FUNCTION_BLOCK FB_EventsManager
VAR_INPUT
    // Presentation-only warning classification; does not request Fault/Stop.
    aWarningEvents : ARRAY[0..4, 0..100] OF BOOL;
	bPulse					: BOOL;
	bDataWritedInCSV		: BOOL;
	nArraySize				: DINT;
	bMachineMessage			: STRING;
	eMachineState 			: E_MachineState;
END_VAR
VAR_OUTPUT
    bMachineFault            : BOOL;
    bCycleStopRequest        : BOOL;
    sSystemDate              : STRING(10);
    sSystemTime              : STRING(8);
	astActiveEvents			: ARRAY [0..50] OF ST_ActiveEvents;
	astEventsHistory		: ARRAY[0..200] OF ST_EventsHistory;
END_VAR
VAR
    aWarningConditionSeen : ARRAY[0..4, 0..100] OF BOOL;
	i								: ARRAY [0..1] OF DINT;
	j								: ARRAY [0..1] OF DINT;
	m								: ARRAY [0..3] OF DINT;
	k								: ARRAY [0..1] OF DINT;
	l								: DINT;
	n								: DINT;
	
	bEventsAssigmentSignal			: BOOL		:= TRUE;
    bStationFaultCondition   : BOOL;
    bStationStopCondition    : BOOL;

    // Local IPC clock used internally for event-history timestamps.
    fbLocalSystemTime        : FB_LocalSystemTime;
END_VAR

VAR_IN_OUT
	
	stStationEvents			: ARRAY[0..4] OF ST_StationEvents;
	stEventsAssigment		: ST_EventsAssigmentGeneral;
	bResetFaults			: BOOL;
	
END_VAR

UpdateSystemDateTime();

ACT_FaultTrig();

ACT_EventTextAssigment();

ACT_ActiveEvents_DataHistory();

// Row zero is permanently reserved for the operational instruction.
astActiveEvents[0].sEventTex := bMachineMessage;
astActiveEvents[0].sType := 'Message';
astActiveEvents[0].abType := 3;
astActiveEvents[0].sSolution := '';

ACTION ACT_ActiveEvents_DataHistory:
// ============================================================================
// ACTIVE EVENTS AND EVENT HISTORY
// ============================================================================
//
// astActiveEvents[0]:
//     Reserved exclusively for the current machine message.
//
// astActiveEvents[1..50]:
//     Active Faults and Cycle Stop Requests.
//
// astEventsHistory:
//     Complete event history.
//
// EVENT BEHAVIOUR:
//
// MESSAGE:
//     - Operator instruction.
//     - Displayed only through astActiveEvents[0].
//     - Never added to rows 1..50.
//
// FAULT:
//     - Latched individually through bActive.
//     - Displayed only while the machine is in Fault.
//     - Remains latched after the live condition disappears.
//     - Cleared by Reset only after bEventFlag is FALSE.
//
// CYCLE STOP REQUEST:
//     - Latched individually through bActive.
//     - Displayed in any machine state.
//     - Remains visible after the live condition disappears.
//     - Cleared by Reset only after bEventFlag is FALSE.
//
// bEventFlag:
//     Live condition.
//
// bActive:
//     Individual event presentation latch.
//
// ============================================================================


IF bPulse THEN

    // ------------------------------------------------------------------------
    // REBUILD ACTIVE EVENT GRID
    // ------------------------------------------------------------------------
    // Row 0 is intentionally preserved because it contains the current
    // machine instruction/message.
    // ------------------------------------------------------------------------

    FOR l := 1 TO 50 DO

        astActiveEvents[l].sEventTex := '';
        astActiveEvents[l].sType := '';
        astActiveEvents[l].abType := 0;
        astActiveEvents[l].sSolution := '';

    END_FOR


    // Rows 1..50 are used for Faults and Alerts.
    l := 0;


    // ------------------------------------------------------------------------
    // SCAN ALL STATION EVENTS
    // ------------------------------------------------------------------------

    FOR k[0] := 0 TO nArraySize DO

        FOR k[1] := 0 TO 100 DO


            // =================================================================
            // FAULT
            // =================================================================

            IF stStationEvents[k[0]].aEvents[k[1]].bFault THEN


                // -------------------------------------------------------------
                // NEW FAULT DETECTED
                // -------------------------------------------------------------
                // Register in history only once, when the live condition
                // activates an event that was not already latched.
                // -------------------------------------------------------------

                IF stStationEvents[k[0]].aEvents[k[1]].bEventFlag
                    AND NOT stStationEvents[k[0]].aEvents[k[1]].bActive
                THEN

                    // Shift history.
                    FOR n := 200 TO 1 BY -1 DO

                        astEventsHistory[n] :=
                            astEventsHistory[n - 1];

                    END_FOR


                    // Insert newest event.
                    astEventsHistory[0].sEventTex :=
                        stStationEvents[k[0]].aEvents[k[1]].bEventTextHMI;

                    astEventsHistory[0].sType :=
                        'Fault';

                    astEventsHistory[0].abType :=
                        1;

                    astEventsHistory[0].sDate :=
                        sSystemDate;

                    astEventsHistory[0].sTime :=
                        sSystemTime;


                    // Latch the individual event.
                    stStationEvents[k[0]].aEvents[k[1]].bActive :=
                        TRUE;

                END_IF


                // -------------------------------------------------------------
                // RESET FAULT LATCH
                // -------------------------------------------------------------
                // Reset is allowed to clear the individual event only after
                // the originating fault condition has disappeared.
                // -------------------------------------------------------------

                IF bResetFaults
                    AND NOT stStationEvents[k[0]].aEvents[k[1]].bEventFlag
                THEN

                    stStationEvents[k[0]].aEvents[k[1]].bActive :=
                        FALSE;

                END_IF


                // -------------------------------------------------------------
                // ACTIVE GRID
                // -------------------------------------------------------------
                // Faults are shown only while the machine itself is in Fault.
                //
                // bActive allows the original cause to remain displayed after
                // bEventFlag has returned FALSE, until the operator resets.
                // -------------------------------------------------------------

                IF stStationEvents[k[0]].aEvents[k[1]].bActive
                    AND eMachineState = E_MachineState.Fault
                THEN

                    IF l < 50 THEN

                        l := l + 1;

                        astActiveEvents[l].sEventTex :=
                            stStationEvents[k[0]].aEvents[k[1]].bEventTextHMI;

                        astActiveEvents[l].sType :=
                            'Fault';

                        astActiveEvents[l].abType :=
                            1;

                        astActiveEvents[l].sSolution :=
                            stStationEvents[k[0]].aEvents[k[1]].sSolution;

                    END_IF

                END_IF



            // =================================================================
            // CYCLE STOP REQUEST / ALERT
            // =================================================================

            ELSIF stStationEvents[k[0]].aEvents[k[1]].bCycleStopRequest THEN


                // -------------------------------------------------------------
                // NEW ALERT DETECTED
                // -------------------------------------------------------------

                IF stStationEvents[k[0]].aEvents[k[1]].bEventFlag
                    AND NOT stStationEvents[k[0]].aEvents[k[1]].bActive
                THEN

                    // Shift history.
                    FOR n := 200 TO 1 BY -1 DO

                        astEventsHistory[n] :=
                            astEventsHistory[n - 1];

                    END_FOR


                    // Insert newest event.
                    astEventsHistory[0].sEventTex :=
                        stStationEvents[k[0]].aEvents[k[1]].bEventTextHMI;

                    astEventsHistory[0].sType :=
                        'Cycle Stop Request';

                    astEventsHistory[0].abType :=
                        2;

                    astEventsHistory[0].sDate :=
                        sSystemDate;

                    astEventsHistory[0].sTime :=
                        sSystemTime;


                    // Latch the individual Alert.
                    stStationEvents[k[0]].aEvents[k[1]].bActive :=
                        TRUE;

                END_IF


                // -------------------------------------------------------------
                // RESET ALERT LATCH
                // -------------------------------------------------------------
                // The Alert remains displayed after the live condition has
                // disappeared and is acknowledged by Reset.
                // -------------------------------------------------------------

                IF bResetFaults
                    AND NOT stStationEvents[k[0]].aEvents[k[1]].bEventFlag
                THEN

                    stStationEvents[k[0]].aEvents[k[1]].bActive :=
                        FALSE;

                END_IF


                // -------------------------------------------------------------
                // ACTIVE GRID
                // -------------------------------------------------------------
                // Alerts may be shown in any machine state.
                // -------------------------------------------------------------

                IF stStationEvents[k[0]].aEvents[k[1]].bActive THEN

                    IF l < 50 THEN

                        l := l + 1;

                        astActiveEvents[l].sEventTex :=
                            stStationEvents[k[0]].aEvents[k[1]].bEventTextHMI;

                        astActiveEvents[l].sType :=
                            'Cycle Stop Request';

                        astActiveEvents[l].abType :=
                            2;

                        astActiveEvents[l].sSolution :=
                            stStationEvents[k[0]].aEvents[k[1]].sSolution;

                    END_IF

                END_IF



            // =================================================================
            // MESSAGE
            // =================================================================
            //
            // Messages are instructions for the operator.
            //
            // They are NOT inserted into astActiveEvents[1..50].
            // Row 0 remains exclusively responsible for the current machine
            // instruction through sMachineMessage.
            //
            // bActive is not used as an operator-reset latch for Messages.
            // =================================================================

            // Resettable warnings use the existing Alert icon (abType=2).
            // The raw condition rearms history; bActive retains display until Reset.
            // Acknowledging a held condition must not re-create the warning.
            ELSIF aWarningEvents[k[0], k[1]] THEN

                IF stStationEvents[k[0]].aEvents[k[1]].bEventFlag
                    AND NOT aWarningConditionSeen[k[0], k[1]]
                THEN
                    FOR n := 200 TO 1 BY -1 DO
                        astEventsHistory[n] := astEventsHistory[n - 1];
                    END_FOR
                    astEventsHistory[0].sEventTex :=
                        stStationEvents[k[0]].aEvents[k[1]].bEventTextHMI;
                    astEventsHistory[0].sType := 'Warning';
                    astEventsHistory[0].abType := 2;
                    astEventsHistory[0].sDate := sSystemDate;
                    astEventsHistory[0].sTime := sSystemTime;
                    stStationEvents[k[0]].aEvents[k[1]].bActive := TRUE;
                END_IF

                aWarningConditionSeen[k[0], k[1]] :=
                    stStationEvents[k[0]].aEvents[k[1]].bEventFlag;
                // Live owner-latched warnings cannot be acknowledged by machine Reset.
                IF stStationEvents[k[0]].aEvents[k[1]].bPersistentMessage THEN
                    stStationEvents[k[0]].aEvents[k[1]].bActive :=
                        stStationEvents[k[0]].aEvents[k[1]].bEventFlag;
                ELSIF bResetFaults THEN
                    stStationEvents[k[0]].aEvents[k[1]].bActive := FALSE;
                END_IF

                IF stStationEvents[k[0]].aEvents[k[1]].bActive AND (l < 50) THEN
                    l := l + 1;
                    astActiveEvents[l].sEventTex :=
                        stStationEvents[k[0]].aEvents[k[1]].bEventTextHMI;
                    astActiveEvents[l].sType := 'Warning';
                    astActiveEvents[l].abType := 2;
                    astActiveEvents[l].sSolution :=
                        stStationEvents[k[0]].aEvents[k[1]].sSolution;
                END_IF

            ELSIF stStationEvents[k[0]].aEvents[k[1]].bMessage THEN


                // -------------------------------------------------------------
                // OPTIONAL MESSAGE HISTORY
                // -------------------------------------------------------------
                // Preserve the existing ability to register message events in
                // history, but rearm them automatically when their condition
                // disappears because Messages do not require operator Reset.
                // -------------------------------------------------------------

                IF stStationEvents[k[0]].aEvents[k[1]].bEventFlag
                    AND NOT stStationEvents[k[0]].aEvents[k[1]].bActive
                THEN

                    FOR n := 200 TO 1 BY -1 DO

                        astEventsHistory[n] :=
                            astEventsHistory[n - 1];

                    END_FOR


                    astEventsHistory[0].sEventTex :=
                        stStationEvents[k[0]].aEvents[k[1]].bEventTextHMI;

                    astEventsHistory[0].sType :=
                        'Message';

                    astEventsHistory[0].abType :=
                        3;

                    astEventsHistory[0].sDate :=
                        sSystemDate;

                    astEventsHistory[0].sTime :=
                        sSystemTime;


                    stStationEvents[k[0]].aEvents[k[1]].bActive :=
                        TRUE;

                END_IF


                // Messages automatically rearm when their live condition ends.
                IF NOT stStationEvents[k[0]].aEvents[k[1]].bEventFlag THEN

                    stStationEvents[k[0]].aEvents[k[1]].bActive :=
                        FALSE;

                END_IF

                // Live message: shown in Active Events while the condition is
                // TRUE and cannot be acknowledged/reset by the operator.
                IF stStationEvents[k[0]].aEvents[k[1]].bPersistentMessage
                    AND stStationEvents[k[0]].aEvents[k[1]].bEventFlag
                THEN

                    IF l < 50 THEN
                        l := l + 1;
                        astActiveEvents[l].sEventTex :=
                            stStationEvents[k[0]].aEvents[k[1]].bEventTextHMI;
                        astActiveEvents[l].sType := 'Message';
                        astActiveEvents[l].abType := 3;
                        astActiveEvents[l].sSolution :=
                            stStationEvents[k[0]].aEvents[k[1]].sSolution;
                    END_IF

                END_IF


            END_IF


        END_FOR

    END_FOR


END_IF
END_ACTION

ACTION ACT_EventTextAssigment:

FOR j[0] := 0 TO nArraySize DO
	
	FOR j[1] := 0 TO 100 DO 
		
		IF stStationEvents[j[0]].aEvents[j[1]].bFault THEN
			
			m[0]											:= m[0]+1;
			
			stStationEvents[j[0]].aEvents[j[1]].bEventTextHMI	:= 		CONCAT( STR1 := 'N ', STR2 := 
																CONCAT( STR1 := DINT_TO_STRING(m[0]), str2 := 
																CONCAT( STR1 :='-Station' , STR2 := 
																CONCAT( STR1 := DINT_TO_STRING(j[0]), STR2 := 
																CONCAT( STR1 :=' - ', str2 := stStationEvents[j[0]].aEvents[j[1]].bEventText )))));
			stStationEvents[j[0]].aEvents[j[1]].bAssignedID	:= 	m[0];				
			
			//EVENTS ASSIGMENT
			stEventsAssigment.astFaultEvents[m[0]].sEventText	:= stStationEvents[j[0]].aEvents[j[1]].bEventTextHMI;
			stEventsAssigment.astFaultEvents[m[0]].sSolution	:= stStationEvents[j[0]].aEvents[j[1]].sSolution;
			
		ELSIF stStationEvents[j[0]].aEvents[j[1]].bCycleStopRequest THEN
		
			m[2]											:= m[2]+1;	
			
			stStationEvents[j[0]].aEvents[j[1]].bEventTextHMI	:= 		CONCAT( STR1 := 'N ', STR2 := 
																CONCAT( STR1 := DINT_TO_STRING(m[2]), str2 := 
																CONCAT( STR1 :='-Station' , STR2 := 
																CONCAT( STR1 := DINT_TO_STRING(j[0]), STR2 := 
																CONCAT( STR1 :=' - ', str2 := stStationEvents[j[0]].aEvents[j[1]].bEventText )))));
			stStationEvents[j[0]].aEvents[j[1]].bAssignedID	:= 	m[2];													

			//EVENTS ASSIGMENT
			stEventsAssigment.astCycleStopRequestEvents[m[2]].sEventText	:= stStationEvents[j[0]].aEvents[j[1]].bEventTextHMI;
			stEventsAssigment.astCycleStopRequestEvents[m[2]].sSolution	:= stStationEvents[j[0]].aEvents[j[1]].sSolution;
			
		ELSIF stStationEvents[j[0]].aEvents[j[1]].bMessage THEN
			
			m[3]											:= m[3]+1;
			
			stStationEvents[j[0]].aEvents[j[1]].bEventTextHMI	:= 		CONCAT( STR1 := 'N ', STR2 := 
																CONCAT( STR1 := DINT_TO_STRING(m[3]), str2 := 
																CONCAT( STR1 :='-Station' , STR2 := 
																CONCAT( STR1 := DINT_TO_STRING(j[0]), STR2 := 
																CONCAT( STR1 :=' - ', str2 := stStationEvents[j[0]].aEvents[j[1]].bEventText )))));
			stStationEvents[j[0]].aEvents[j[1]].bAssignedID	:= 	m[3];													
				
			//EVENTS ASSIGMENT
			stEventsAssigment.astMessage[m[3]].sEventText	:= stStationEvents[j[0]].aEvents[j[1]].bEventTextHMI;
			stEventsAssigment.astMessage[m[3]].sSolution	:= stStationEvents[j[0]].aEvents[j[1]].sSolution;	
			
		END_IF
		
	END_FOR
	
	
END_FOR
j[0]														:= 0;
j[1]														:= 0;
m[0]														:= 0;
m[1]														:= 0;
m[2]														:= 0;
m[3]														:= 0;
END_ACTION

ACTION ACT_FaultTrig:
// Deterministic station aggregation. Classification is fixed in each point;
// bEventFlag is the live condition. Station flags are latched until Reset.
bMachineFault := FALSE;
bCycleStopRequest := FALSE;

FOR i[0] := 0 TO nArraySize DO
    bStationFaultCondition := FALSE;
    bStationStopCondition := FALSE;

    FOR i[1] := 0 TO 100 DO
        bStationFaultCondition := bStationFaultCondition
            OR (stStationEvents[i[0]].aEvents[i[1]].bFault
                AND stStationEvents[i[0]].aEvents[i[1]].bEventFlag);

        bStationStopCondition := bStationStopCondition
            OR (stStationEvents[i[0]].aEvents[i[1]].bCycleStopRequest
                AND stStationEvents[i[0]].aEvents[i[1]].bEventFlag);
    END_FOR

    IF bStationFaultCondition THEN
        stStationEvents[i[0]].bFault := TRUE;
    ELSIF bResetFaults THEN
        stStationEvents[i[0]].bFault := FALSE;
    END_IF

    IF bStationStopCondition THEN
        stStationEvents[i[0]].bCycleStopRequest := TRUE;
    ELSIF bResetFaults THEN
        stStationEvents[i[0]].bCycleStopRequest := FALSE;
    END_IF

    bMachineFault := bMachineFault OR stStationEvents[i[0]].bFault;
    bCycleStopRequest := bCycleStopRequest OR stStationEvents[i[0]].bCycleStopRequest;
END_FOR
END_ACTION

METHOD PRIVATE UpdateSystemDateTime
VAR
END_VAR
// Read the local Windows/IPC clock.
fbLocalSystemTime(
    sNetID := '',
    bEnable := TRUE,
    dwCycle := 5,
    dwOpt := 1,
    tTimeout := T#5S
);

// Date: DD/MM/YYYY
sSystemDate := '';

IF fbLocalSystemTime.systemTime.wDay < 10 THEN
    sSystemDate := CONCAT(sSystemDate, '0');
END_IF

sSystemDate := CONCAT(
    sSystemDate,
    UINT_TO_STRING(fbLocalSystemTime.systemTime.wDay)
);

sSystemDate := CONCAT(sSystemDate, '/');

IF fbLocalSystemTime.systemTime.wMonth < 10 THEN
    sSystemDate := CONCAT(sSystemDate, '0');
END_IF

sSystemDate := CONCAT(
    sSystemDate,
    UINT_TO_STRING(fbLocalSystemTime.systemTime.wMonth)
);

sSystemDate := CONCAT(sSystemDate, '/');

sSystemDate := CONCAT(
    sSystemDate,
    UINT_TO_STRING(fbLocalSystemTime.systemTime.wYear)
);

// Time: HH:MM:SS
sSystemTime := '';

IF fbLocalSystemTime.systemTime.wHour < 10 THEN
    sSystemTime := CONCAT(sSystemTime, '0');
END_IF

sSystemTime := CONCAT(
    sSystemTime,
    UINT_TO_STRING(fbLocalSystemTime.systemTime.wHour)
);

sSystemTime := CONCAT(sSystemTime, ':');

IF fbLocalSystemTime.systemTime.wMinute < 10 THEN
    sSystemTime := CONCAT(sSystemTime, '0');
END_IF

sSystemTime := CONCAT(
    sSystemTime,
    UINT_TO_STRING(fbLocalSystemTime.systemTime.wMinute)
);

sSystemTime := CONCAT(sSystemTime, ':');

IF fbLocalSystemTime.systemTime.wSecond < 10 THEN
    sSystemTime := CONCAT(sSystemTime, '0');
END_IF

sSystemTime := CONCAT(
    sSystemTime,
    UINT_TO_STRING(fbLocalSystemTime.systemTime.wSecond)
);
END_METHOD

END_FUNCTION_BLOCK

(* stored: Version 1.1.0.1, ProductVersion 3.1.4026.18
   POU FB_EventsManager: Id {9ecba55d-bb6b-489e-b76b-d005a96f9d84}, SpecialFunc None
   Action ACT_ActiveEvents_DataHistory: Id {61da313d-b258-4798-832e-c39696bf6052}
   Action ACT_EventTextAssigment: Id {0dfbbd34-04a8-4fd4-a700-4471e514f320}
   Action ACT_FaultTrig: Id {68bdf7df-b8fd-4397-a284-4a9760510255}
   Method UpdateSystemDateTime: Id {14a21f98-57c6-4a84-a16e-d3b4abaff015} *)
